{attribute 'pack_mode':='1'}
TYPE HeartbeatParams :
STRUCT
   current_time_ms : ULINT; (* Current time in milliseconds from the
overarching system. *)
END_STRUCT
END_TYPE

(* stored: Version 1.1.0.1, ProductVersion 3.1.4024.12
   DUT HeartbeatParams: Id {822ee884-be1b-40dd-b166-a82cddfc47ab} *)
